FUNCTION_BLOCK "Convention23"
TITLE = Test for rule Convention 23




VAR_INPUT
bla : Any; // OK
END_VAR
VAR_IN_OUT
foo : Any; // Violation
// some extra comments
bar: Any; // Violation
END_VAR
BEGIN
END_FUNCTION_BLOCK
